Fanuc KAREL source: kd00029.KL

-- PROVISIONAL review KL for V1013-1; original PC SHA256 8b83ce28527be74580c20eb480957f041391a7384738294b6d69bff94b0f65f9
-- Incomplete behavior may be omitted. Consult companion uncertainty JSON. Do not deploy.
PROGRAM KD00029
%NOLOCKGROUP
VAR
  I : INTEGER
  J : INTEGER
  B : BOOLEAN
  R : REAL
  S : STRING[80]
BEGIN
  -- UNRESOLVED_PC offsets 5-21; opcodes 9D,81,18,9C,12,22,9D,13,04
  -- UNRESOLVED_PC offsets 26-30; opcodes 7F
END KD00029
